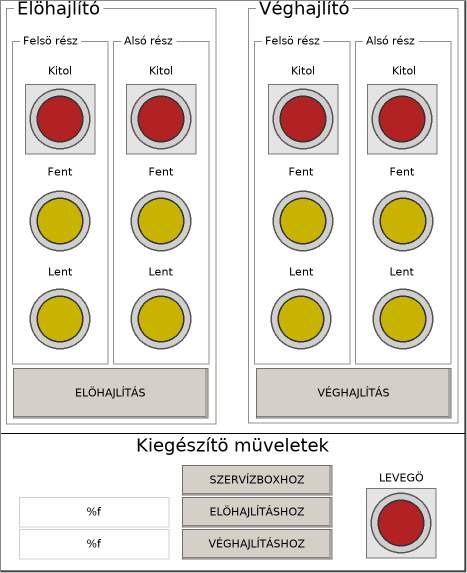
VISUALIZATION Hajlitok  // 467x573
    Rectangle (0,0 465x571)
    GroupBox (6,0 210x424), "Elöhajlító"
        GroupBox (6,33 96x331), "Felsö rész"
            PushSwitch (13,51 70x70), variable: HAJLITOK.bElohajlitoFelso, behaviour: TOGGLE, style: Switch-PushSwitch-Red
            Label (14,23 68x30), "Kitol"
            Lamp1 (13,153 70x70), variable: HAJLITOK.bElohajlitoFelsoFent, style: Lamp-Lamp1-Yellow
            Label (27,124 42x30), "Fent"
            Lamp1 (13,251 70x70), variable: HAJLITOK.bElohajlitoFelsoLent, style: Lamp-Lamp1-Yellow
            Label (29,224 39x30), "Lent"
        GroupBox (107,33 96x331), "Alsó rész"
            Label (14,23 68x30), "Kitol"
            Label (27,124 42x30), "Fent"
            PushSwitch (13,51 70x70), variable: HAJLITOK.bElohajlitoAlso, behaviour: TOGGLE, style: Switch-PushSwitch-Red
            Lamp1 (13,153 70x70), variable: HAJLITOK.bElohajlitoAlsoFent, style: Lamp-Lamp1-Yellow
            Lamp1 (13,251 70x70), variable: HAJLITOK.bElohajlitoAlsoLent, style: Lamp-Lamp1-Yellow
            Label (28,224 40x30), "Lent"
        Button (7,368 195x50), "ELÖHAJLÍTÁS", input disabled if: HAJLITOK.s_InCommand <> ''
            OnMouseUp: execute {
                IF HAJLITOK.s_InCommand = '' THEN
                	HAJLITOK.s_InCommand:='ELOHAJLITAS';
                END_IF
            }
    GroupBox (248,0 210x423), "Véghajlító"
        GroupBox (6,33 96x331), "Felsö rész"
            Label (15,23 68x30), "Kitol"
            Label (26,124 42x30), "Fent"
            Label (28,224 39x30), "Lent"
            PushSwitch (14,51 70x70), variable: HAJLITOK.bVeghajlitoFelso, behaviour: TOGGLE, style: Switch-PushSwitch-Red
            Lamp1 (14,153 70x70), variable: HAJLITOK.bVeghajlitoFelsoFent, style: Lamp-Lamp1-Yellow
            Lamp1 (12,251 70x70), variable: HAJLITOK.bVeghajlitoFelsoLent, style: Lamp-Lamp1-Yellow
        GroupBox (107,33 96x331), "Alsó rész"
            Label (15,23 68x30), "Kitol"
            Label (26,124 42x30), "Fent"
            Label (27,224 40x30), "Lent"
            PushSwitch (12,51 70x70), variable: HAJLITOK.bVeghajlitoAlso, behaviour: TOGGLE, style: Switch-PushSwitch-Red
            Lamp1 (13,153 70x70), variable: HAJLITOK.bVeghajlitoAlsoFent, style: Lamp-Lamp1-Yellow
            Lamp1 (13,251 70x70), variable: HAJLITOK.bVeghajlitoAlsoLent, style: Lamp-Lamp1-Yellow
        Button (8,368 195x50), "VÉGHAJLÍTÁS", input disabled if: HAJLITOK.s_InCommand <> ''
            OnMouseUp: execute {
                IF HAJLITOK.s_InCommand = '' THEN
                	HAJLITOK.s_InCommand:='VEGHAJLITAS';
                END_IF
            }
    Line (0,433) (465,433), "Kiegészítö müveletek"
    Textfield (19,497 150x30), "%f", text variable: GVL.lrHajlitoPosition1
        OnMouseClick: write the text variable via VisuDialogs.Numpad, min -10000, max -1
    Button (182,497 150x30), "ELÖHAJLÍTÁSHOZ", text variable: GVL.lrHajlitoPosition1
        OnMouseUp: execute { JOZSITENGELY.lrJozsiPosition:=GVL.lrHajlitoPosition1; JOZSITENGELY.sJozsiAxisCommand:='MOVE'; }
    Textfield (19,529 150x30), "%f", text variable: GVL.lrHajlitoPosition2
        OnMouseClick: write the text variable via VisuDialogs.Numpad, min -10000, max -1
    Button (182,529 150x30), "VÉGHAJLÍTÁSHOZ"
        OnMouseUp: execute { JOZSITENGELY.lrJozsiPosition:=GVL.lrHajlitoPosition2; JOZSITENGELY.sJozsiAxisCommand:='MOVE'; }
    Button (182,465 150x30), "SZERVÍZBOXHOZ"
        OnMouseUp: execute { JOZSITENGELY.lrJozsiPosition:=GVL.lrNTCSzervizbox; JOZSITENGELY.sJozsiAxisCommand:='MOVE'; }
    Group (366,463 70x95)
        PushSwitch (0,25 70x70), variable: MAIN.bLevego, behaviour: TOGGLE, style: Switch-PushSwitch-Red
        Label (1,0 69x30), "LEVEGÖ"
END_VISUALIZATION

(* stored: Version 1.1.0.1, ProductVersion 3.1.4024.11
   Visu Hajlitok: Id {911f360f-597a-4b73-8a42-c2bf1f7f8ad1} *)
